PROGRAM Mod103
VAR
	IO_f : ARRAY [1..16] OF IO_force;
	i: SINT;
END_VAR

	// 輸入模組1
	FOR i := 1 TO 16 DO
		IO_f[i](Raw_IO := EtherCAT.MainMod_3.Input[i], Out =>MainIO.io103.In[i]);
	END_FOR
	
	
	MainIO.io103_s.0 := IO_f[1].Out;
	MainIO.io103_s.1 := IO_f[2].Out;
	MainIO.io103_s.2 := IO_f[3].Out;
	MainIO.io103_s.3 := IO_f[4].Out;
	MainIO.io103_s.4 := IO_f[5].Out;
	MainIO.io103_s.5 := IO_f[6].Out;
	MainIO.io103_s.6 := IO_f[7].Out;
	MainIO.io103_s.7 := IO_f[8].Out;
	MainIO.io103_s.8 := IO_f[9].Out;
	MainIO.io103_s.9 := IO_f[10].Out;
	MainIO.io103_s.10 := IO_f[11].Out;
	MainIO.io103_s.11 := IO_f[12].Out;
	MainIO.io103_s.12 := IO_f[13].Out;
	MainIO.io103_s.13 := IO_f[14].Out;
	MainIO.io103_s.14 := IO_f[15].Out;
	MainIO.io103_s.15 := IO_f[16].Out;
	
	MainIO.io103_f.0 := IO_f[1].ForceEnable;
	MainIO.io103_f.1 := IO_f[2].ForceEnable;
	MainIO.io103_f.2 := IO_f[3].ForceEnable;
	MainIO.io103_f.3 := IO_f[4].ForceEnable;
	MainIO.io103_f.4 := IO_f[5].ForceEnable;
	MainIO.io103_f.5 := IO_f[6].ForceEnable;
	MainIO.io103_f.6 := IO_f[7].ForceEnable;
	MainIO.io103_f.7 := IO_f[8].ForceEnable;
	MainIO.io103_f.8 := IO_f[9].ForceEnable;
	MainIO.io103_f.9 := IO_f[10].ForceEnable;
	MainIO.io103_f.10 := IO_f[11].ForceEnable;
	MainIO.io103_f.11 := IO_f[12].ForceEnable;
	MainIO.io103_f.12 := IO_f[13].ForceEnable;
	MainIO.io103_f.13 := IO_f[14].ForceEnable;
	MainIO.io103_f.14 := IO_f[15].ForceEnable;
	MainIO.io103_f.15 := IO_f[16].ForceEnable;

END_PROGRAM

(* stored: Version 1.1.0.1, ProductVersion 3.1.4024.15
   POU Mod103: Id {618b947a-e142-4dfb-8905-23468095ce66}, SpecialFunc None *)
